// Mitsubishi GX Works2 project: EX01   PLC: Q03UD

PROGRAM MAIN
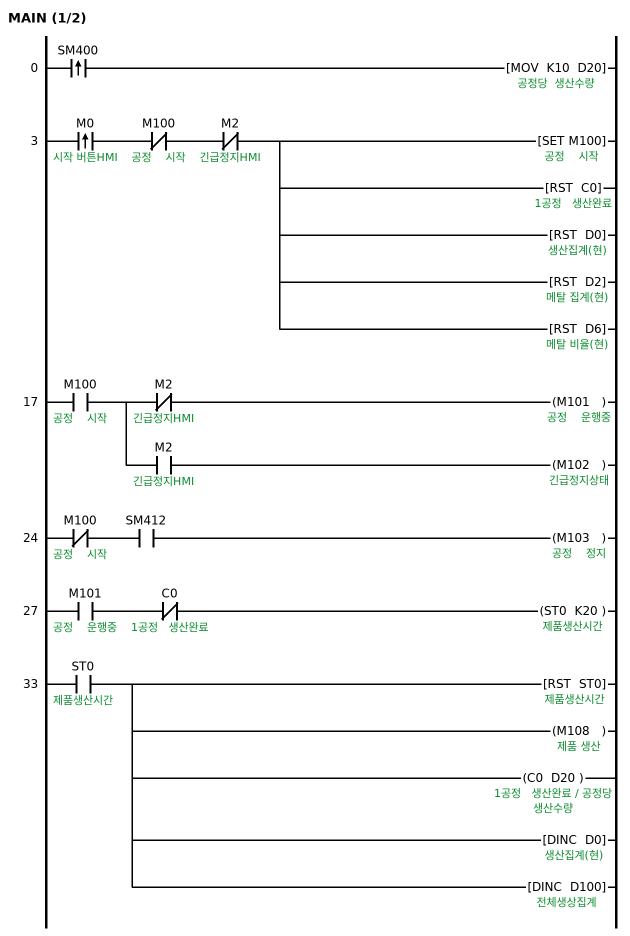
0     LDP     SM400
      MOV     K10 D20  ; 공정당  생산수량
3     LDP     M0  ; 시작 버튼HMI
      ANI     M100  ; 공정    시작
      ANI     M2  ; 긴급정지HMI
      SET     M100  ; 공정    시작
      RST     C0  ; 1공정   생산완료
      RST     D0  ; 생산집계(현)
      RST     D2  ; 메탈 집계(현)
      RST     D6  ; 메탈 비율(현)
17    LD      M100  ; 공정    시작
      MPS
      ANI     M2  ; 긴급정지HMI
      OUT     M101  ; 공정    운행중
      MPP
      AND     M2  ; 긴급정지HMI
      OUT     M102  ; 긴급정지상태
24    LDI     M100  ; 공정    시작
      AND     SM412
      OUT     M103  ; 공정    정지
27    LD      M101  ; 공정    운행중
      ANI     C0  ; 1공정   생산완료
      OUT     ST0 K20  ; 제품생산시간
33    LD      ST0  ; 제품생산시간
      RST     ST0  ; 제품생산시간
      OUT     M108  ; 제품 생산
      OUT     C0 D20  ; 1공정   생산완료 / 공정당  생산수량
      DINC    D0
      DINC    D100  ; 전체생상집계
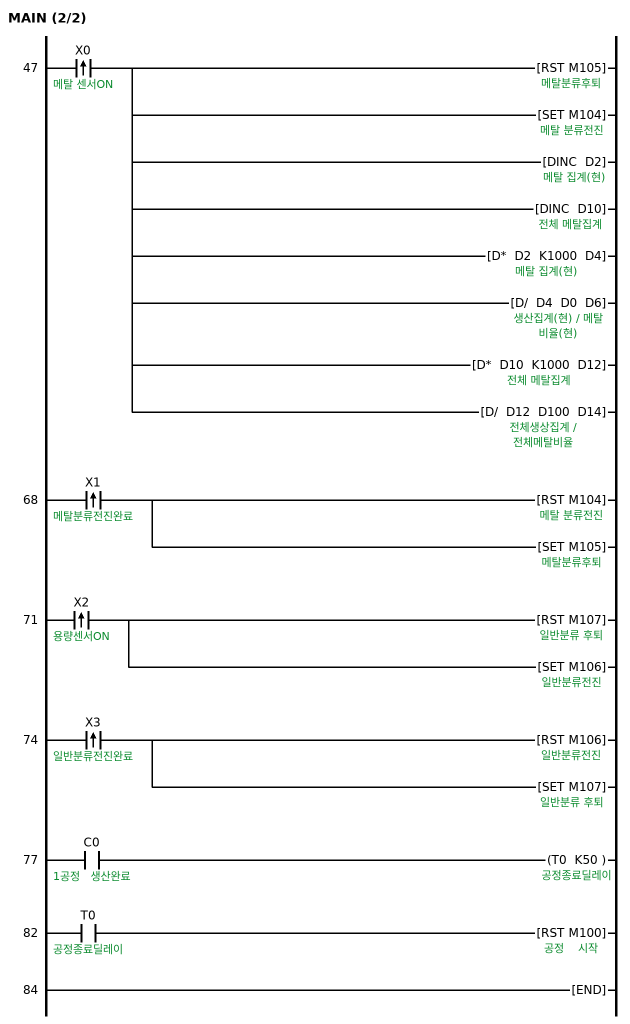
47    LDP     X0  ; 메탈 센서ON
      RST     M105  ; 메탈분류후퇴
      SET     M104  ; 메탈 분류전진
      DINC    D2
      DINC    D10  ; 전체 메탈집계
      D*      D2 K1000 D4
      D/      D4 D0 D6
      D*      D10 K1000 D12
      D/      D12 D100 D14  ; 전체메탈비율
68    LDP     X1  ; 메탈분류전진완료
      RST     M104  ; 메탈 분류전진
      SET     M105  ; 메탈분류후퇴
71    LDP     X2  ; 용량센서ON
      RST     M107  ; 일반분류 후퇴
      SET     M106  ; 일반분류전진
74    LDP     X3  ; 일반분류전진완료
      RST     M106  ; 일반분류전진
      SET     M107  ; 일반분류 후퇴
77    LD      C0  ; 1공정   생산완료
      OUT     T0 K50  ; 공정종료딜레이
82    LD      T0  ; 공정종료딜레이
      RST     M100  ; 공정    시작
84    END
END_PROGRAM

PROGRAM OUTPUT
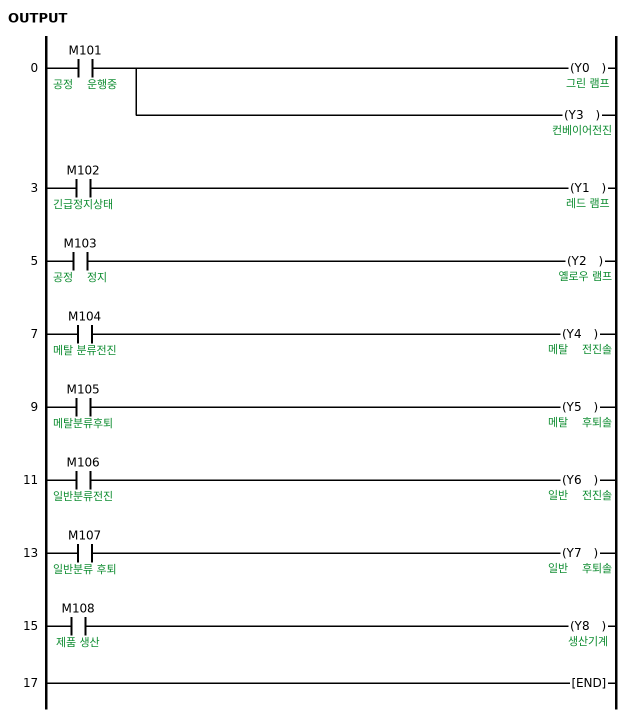
0     LD      M101  ; 공정    운행중
      OUT     Y0  ; 그린 램프
      OUT     Y3  ; 컨베이어전진
3     LD      M102  ; 긴급정지상태
      OUT     Y1  ; 레드 램프
5     LD      M103  ; 공정    정지
      OUT     Y2  ; 옐로우 램프
7     LD      M104  ; 메탈 분류전진
      OUT     Y4  ; 메탈    전진솔
9     LD      M105  ; 메탈분류후퇴
      OUT     Y5  ; 메탈    후퇴솔
11    LD      M106  ; 일반분류전진
      OUT     Y6  ; 일반    전진솔
13    LD      M107  ; 일반분류 후퇴
      OUT     Y7  ; 일반    후퇴솔
15    LD      M108  ; 제품 생산
      OUT     Y8  ; 생산기계
17    END
END_PROGRAM

// device comments not shown above
M1  ; 정지 버튼HMI
D8  ; 전체생산집계
